(* PLC project Untitled1, Beckhoff Automation GmbH TwinCAT PLC Control 3.5.13.21 *)
(* stored: creationDateTime 2023-11-18T11:54:06.5386523, modificationDateTime 2023-11-18T11:54:06.545484 *)

{attribute 'qualified_only'}
{attribute 'strict'}
TYPE E_Shape :
(
	init := 0,
	Circle,
	Rectangle,
	Sqaure,
	Star,
	Triangle,
	end,
	Custom
);
END_TYPE

INTERFACE I_Shape
METHOD M_Draw : BOOL
VAR_INPUT
END_VAR
END_METHOD
END_INTERFACE

{attribute 'hide_all_locals'}
FUNCTION_BLOCK FB_ShapeCreator
VAR_INPUT
	eShape : E_Shape;
END_VAR
VAR_OUTPUT
END_VAR
VAR
      pCircle    : POINTER TO FB_Circle;
      pRectangle : POINTER TO FB_Rectangle;
      pSquare    : POINTER TO FB_Square;
      pStar      : POINTER TO FB_Star;
      pTriangle  : POINTER TO FB_Triangle;
      iShape 	 : I_Shape;
END_VAR

                  //Hemos declarado punteros a cada bloque de función de forma correspondiente, 
//lo que nos permitiría crear una instancia dinámica del bloque de función de forma solicitado y ahorrar espacio en la memoria. 
//Si los hubiéramos declarado como fbCircle : FB_Circle en su lugar y asumiéramos que nunca necesitaríamos dibujar Circle, 
//aún ocuparíamos el espacio de memoria en este bloque de funciones. 

//En el programa principal, el usuario proporcionará una entrada para la forma deseada y 'M_GetShapeObject' decidirá qué bloque de función de forma crear una instancia y lo devolverá. 
                

METHOD FB_exit : BOOL
VAR_INPUT
	bInCopyCode : BOOL; // if TRUE, the exit method is called for exiting an instance that is copied afterwards (online change).
END_VAR
                        IF (pCircle <> 0) THEN
  __DELETE(pCircle);
  pCircle := 0;
END_IF

IF (pRectangle <> 0) THEN
  __DELETE(pRectangle);
  pRectangle := 0;
END_IF

IF (pSquare <> 0) THEN
  __DELETE(pSquare);
  pSquare := 0;
END_IF

IF (pStar <> 0) THEN
  __DELETE(pStar);
  pStar := 0;
END_IF

IF (pTriangle <> 0) THEN
  __DELETE(pTriangle);
  pTriangle := 0;
END_IF
                      
END_METHOD

METHOD M_GetShapeObject : I_shape
VAR_INPUT
END_VAR
                        CASE eShape OF
	E_Shape.Circle:
		
		//Dynamic instantiation  
		pCircle := __NEW(FB_Circle);
		iShape := pCircle^;
		
		//Return the object
		IF iShape <> 0 THEN
			M_GetShapeObject := iShape;
		END_IF
		
		//Release the memory
		IF (pCircle <> 0) THEN
			__DELETE(pCircle);
			pCircle := 0;
		END_IF
		
		eShape := E_Shape.init;
	
	E_Shape.Rectangle:
		pRectangle := __NEW(FB_Rectangle);
		iShape := pRectangle^;
		
		//Return the object
		IF iShape <> 0 THEN
			M_GetShapeObject := iShape;
		END_IF
		
		IF (pRectangle <> 0) THEN
			__DELETE(pRectangle);
			pRectangle := 0;
		END_IF
		
		eShape := E_Shape.init;	
		
	E_Shape.Sqaure:
		pSquare := __NEW(FB_Square);
		iShape := pSquare^;
		
		//Return the object
		IF iShape <> 0 THEN
			M_GetShapeObject := iShape;
		END_IF
		
		IF (pSquare <> 0) THEN
			__DELETE(pSquare);
			pSquare := 0;
		END_IF
		
		eShape := E_Shape.init;	

	E_Shape.Star:
		pStar := __NEW(FB_Star);
		iShape := pStar^;
		
		//Return the object
		IF iShape <> 0 THEN
			M_GetShapeObject := iShape;
		END_IF
		
		IF (pStar <> 0) THEN
			__DELETE(pStar);
			pStar := 0;
		END_IF
		
		eShape := E_Shape.init;	
	
	E_Shape.Triangle:
		pTriangle := __NEW(FB_Triangle);
		iShape := pTriangle^;
		
		//Return the object
		IF iShape <> 0 THEN
			M_GetShapeObject := iShape;
		END_IF
		
		IF (pTriangle <> 0) THEN
			__DELETE(pTriangle);
			pTriangle := 0;
		END_IF
		
		eShape := E_Shape.init;	
END_CASE
                      
END_METHOD

METHOD M_ReleaseMemory : BOOL
VAR_INPUT
END_VAR
                        IF (pCircle <> 0) THEN
  __DELETE(pCircle);
  pCircle := 0;
END_IF

IF (pRectangle <> 0) THEN
  __DELETE(pRectangle);
  pRectangle := 0;
END_IF

IF (pSquare <> 0) THEN
  __DELETE(pSquare);
  pSquare := 0;
END_IF

IF (pStar <> 0) THEN
  __DELETE(pStar);
  pStar := 0;
END_IF

IF (pTriangle <> 0) THEN
  __DELETE(pTriangle);
  pTriangle := 0;
END_IF
                      
END_METHOD
END_FUNCTION_BLOCK

FUNCTION_BLOCK FB_ShapeCreatorEX EXTENDS FB_ShapeCreator
VAR_INPUT
END_VAR
VAR_OUTPUT
END_VAR
VAR
	pCustomShape : POINTER TO FB_CustomShape;
END_VAR

                  
                

METHOD M_GetShapeObject : I_shape
VAR_INPUT
END_VAR
                        IF eShape = E_Shape.Custom THEN
	
	//Dynamic instantiation  
	pCustomShape := __NEW(FB_CustomShape);
	iShape := pCustomShape^;
	
	//Return the object
	IF iShape <> 0 THEN
		M_GetShapeObject := iShape;
	END_IF
	
	//Release the memory
	IF (pCustomShape <> 0) THEN
		__DELETE(pCustomShape);
		pCustomShape := 0;
	END_IF
	
	eShape := E_Shape.init;
ELSE
	M_GetShapeObject := SUPER^.M_GetShapeObject();
END_IF
                      
END_METHOD
END_FUNCTION_BLOCK

PROGRAM MAIN
VAR
//	fbShapeCreator : FB_ShapeCreator;
	fbShapeCreator : FB_ShapeCreatorEX;
	eShape : E_Shape := E_Shape.init;
	
	iShape : I_Shape;
END_VAR

                  fbShapeCreator(eShape:= eShape);

CASE eShape OF
	E_Shape.Circle:
		iShape := fbShapeCreator.M_GetShapeObject();
		IF iShape <> 0 THEN
			iShape.M_Draw();
		END_IF	
	
		eShape := E_Shape.Rectangle;
	
	E_Shape.Rectangle:
		iShape := fbShapeCreator.M_GetShapeObject();
		IF iShape <> 0 THEN
			iShape.M_Draw();
		END_IF
		
		eShape := E_Shape.Sqaure;	
		
	E_Shape.Sqaure:
		iShape := fbShapeCreator.M_GetShapeObject();
		IF iShape <> 0 THEN
			iShape.M_Draw();
		END_IF	
	
		eShape := E_Shape.Star;	

	E_Shape.Star:
		iShape := fbShapeCreator.M_GetShapeObject();
		IF iShape <> 0 THEN
			iShape.M_Draw();
		END_IF
		
		eShape := E_Shape.Triangle;	
	
	E_Shape.Triangle:
		iShape := fbShapeCreator.M_GetShapeObject();
		IF iShape <> 0 THEN
			iShape.M_Draw();
		END_IF	
	
		//eShape := E_Shape.end;	
		eShape := E_Shape.Custom;	
		
	E_Shape.Custom:
		iShape := fbShapeCreator.M_GetShapeObject();
		IF iShape <> 0 THEN
			iShape.M_Draw();
		END_IF
		
		eShape := E_Shape.end;	
END_CASE
                
END_PROGRAM

{attribute 'enable_dynamic_creation'}
FUNCTION_BLOCK FB_Circle IMPLEMENTS I_Shape
VAR_INPUT
END_VAR
VAR_OUTPUT
END_VAR
VAR
END_VAR

                  //Agregue el {atributo 'enable_dynamic_creation'} en la parte superior de la sección de declaración de cada bloque de funciones. 
//Esto nos permitirá crear una instancia de cada bloque de funciones dinámicamente usando el operador _NEW en el bloque de funciones FB_ShapeCreator. 
                

METHOD M_Draw : BOOL
                        ADSLOGSTR(ADSLOG_MSGTYPE_HINT, 'Draw circle', '');
M_Draw := TRUE;
                      
END_METHOD
END_FUNCTION_BLOCK

{attribute 'enable_dynamic_creation'} 
FUNCTION_BLOCK FB_CustomShape IMPLEMENTS I_Shape
VAR_INPUT
END_VAR
VAR_OUTPUT
END_VAR
VAR
END_VAR

                  
                

{warning 'Agregar implementación de método'}
METHOD M_Draw : BOOL
                        ADSLOGSTR(ADSLOG_MSGTYPE_HINT, 'Draw custom shape', '');
M_Draw := TRUE;
                      
END_METHOD
END_FUNCTION_BLOCK

{attribute 'enable_dynamic_creation'}
FUNCTION_BLOCK FB_Rectangle IMPLEMENTS I_Shape
VAR_INPUT
END_VAR
VAR_OUTPUT
END_VAR
VAR
END_VAR

                  
                

{warning 'Agregar implementación de método'}
METHOD M_Draw : BOOL
                        ADSLOGSTR(ADSLOG_MSGTYPE_HINT, 'Draw rectangle', '');
M_Draw := TRUE;
                      
END_METHOD
END_FUNCTION_BLOCK

{attribute 'enable_dynamic_creation'}
FUNCTION_BLOCK FB_Square IMPLEMENTS I_Shape
VAR_INPUT
END_VAR
VAR_OUTPUT
END_VAR
VAR
END_VAR

                  
                

{warning 'Agregar implementación de método'}
METHOD M_Draw : BOOL
                        ADSLOGSTR(ADSLOG_MSGTYPE_HINT, 'Square', '');
M_Draw := TRUE;
                      
END_METHOD
END_FUNCTION_BLOCK

{attribute 'enable_dynamic_creation'}
FUNCTION_BLOCK FB_Star IMPLEMENTS I_Shape
VAR_INPUT
END_VAR
VAR_OUTPUT
END_VAR
VAR
END_VAR

                  
                

{warning 'Agregar implementación de método'}
METHOD M_Draw : BOOL
                        ADSLOGSTR(ADSLOG_MSGTYPE_HINT, 'Draw Star', '');
M_Draw := TRUE;
                      
END_METHOD
END_FUNCTION_BLOCK

{attribute 'enable_dynamic_creation'}
FUNCTION_BLOCK FB_Triangle IMPLEMENTS I_Shape
VAR_INPUT
END_VAR
VAR_OUTPUT
END_VAR
VAR
END_VAR

                  
                

{warning 'Agregar implementación de método'}
METHOD M_Draw : BOOL
                        ADSLOGSTR(ADSLOG_MSGTYPE_HINT, 'Draw Triangle', '');
M_Draw := TRUE;
                      
END_METHOD
END_FUNCTION_BLOCK

CONFIGURATION Application
  RESOURCE Untitled1 ON PLC
    TASK PlcTask(INTERVAL := T#0ms, PRIORITY := 20);
    PROGRAM MAIN WITH PlcTask : MAIN;
  END_RESOURCE
END_CONFIGURATION
